KUKA KRL program: LOGO.src, LOGO.dat

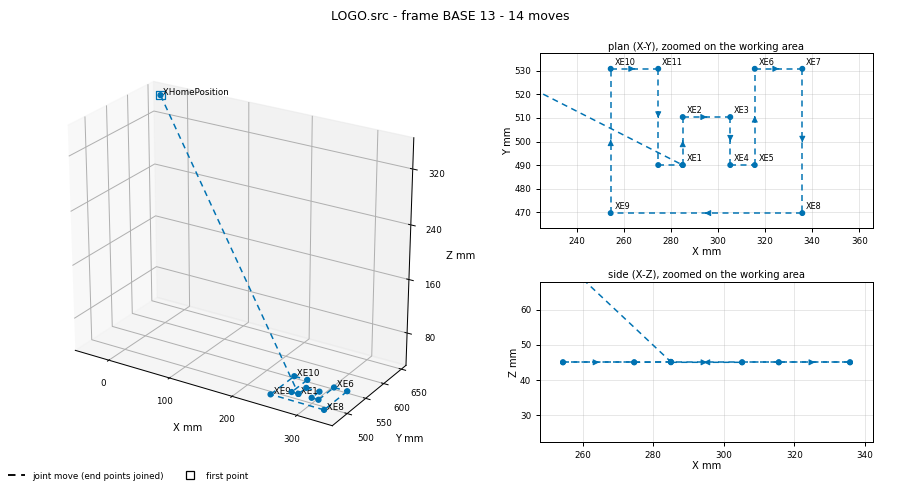
[picture p0: tool path of LOGO.src in frame BASE 13, 14 of 14 moves have a stored position in this frame; points joined in program order, loops and branches not executed]
--- LOGO.src ---
&ACCESS RVP
&REL 3
&PARAM EDITMASK = *
&PARAM TEMPLATE = C:\KRC\Roboter\Template\vorgabe

DEF LOGO( )
;FOLD INI;%{PE}
  ;FOLD BASISTECH INI
    GLOBAL INTERRUPT DECL 3 WHEN $STOPMESS==TRUE DO IR_STOPM ( )
    INTERRUPT ON 3
    BAS (#INITMOV,0 )
  ;ENDFOLD (BASISTECH INI)
  ;FOLD USER INI
    ;Make your modifications here

  ;ENDFOLD (USER INI)
;ENDFOLD (INI)


$BWDSTART=FALSE
PDAT_ACT=PPDAT1
FDAT_ACT=FHomePosition
BAS(#PTP_PARAMS,100)
PTP XHomePosition

$BWDSTART=FALSE
PDAT_ACT=PPDAT1
FDAT_ACT=FE1
BAS(#PTP_PARAMS,100)
PTP XE1
$BWDSTART=FALSE
PDAT_ACT=PPDAT1
FDAT_ACT=FE1
BAS(#PTP_PARAMS,100)
PTP XE2
$BWDSTART=FALSE
PDAT_ACT=PPDAT1
FDAT_ACT=FE1
BAS(#PTP_PARAMS,100)
PTP XE3
$BWDSTART=FALSE
PDAT_ACT=PPDAT1
FDAT_ACT=FE1
BAS(#PTP_PARAMS,100)
PTP XE4
$BWDSTART=FALSE
PDAT_ACT=PPDAT1
FDAT_ACT=FE1
BAS(#PTP_PARAMS,100)
PTP XE5
$BWDSTART=FALSE
PDAT_ACT=PPDAT1
FDAT_ACT=FE1
BAS(#PTP_PARAMS,100)
PTP XE6
$BWDSTART=FALSE
PDAT_ACT=PPDAT1
FDAT_ACT=FE1
BAS(#PTP_PARAMS,100)
PTP XE7
$BWDSTART=FALSE
PDAT_ACT=PPDAT1
FDAT_ACT=FE1
BAS(#PTP_PARAMS,100)
PTP XE8
$BWDSTART=FALSE
PDAT_ACT=PPDAT1
FDAT_ACT=FE1
BAS(#PTP_PARAMS,100)
PTP XE9
$BWDSTART=FALSE
PDAT_ACT=PPDAT1
FDAT_ACT=FE1
BAS(#PTP_PARAMS,100)
PTP XE10
$BWDSTART=FALSE
PDAT_ACT=PPDAT1
FDAT_ACT=FE1
BAS(#PTP_PARAMS,100)
PTP XE11
$BWDSTART=FALSE
PDAT_ACT=PPDAT1
FDAT_ACT=FE1
BAS(#PTP_PARAMS,100)
PTP XE12
$BWDSTART=FALSE
PDAT_ACT=PPDAT1
FDAT_ACT=FE1
BAS(#PTP_PARAMS,100)
PTP XE1
; Offset
;PTP {X 0,Y 0,Z 50,A 0,B 0,C 0} : XE1

END

--- LOGO.dat ---
&ACCESS RVP
&REL 3
&PARAM EDITMASK = *
&PARAM TEMPLATE = C:\KRC\Roboter\Template\vorgabe
DEFDAT  LOGO
;FOLD EXTERNAL DECLARATIONS;%{PE}%MKUKATPBASIS,%CEXT,%VCOMMON,%P
;FOLD BASISTECH EXT;%{PE}%MKUKATPBASIS,%CEXT,%VEXT,%P
EXT  BAS (BAS_COMMAND  :IN,REAL  :IN )
DECL INT SUCCESS
;ENDFOLD (BASISTECH EXT)
;FOLD USER EXT;%{E}%MKUKATPUSER,%CEXT,%VEXT,%P
;Make your modifications here

;ENDFOLD (USER EXT)
;ENDFOLD (EXTERNAL DECLARATIONS)
DECL BASIS_SUGG_T LAST_BASIS={POINT1[] "E12                      ",POINT2[] "E12                      ",CP_PARAMS[] "CPDAT0                  ",PTP_PARAMS[] "PDAT1                   ",CONT[] "                        ",CP_VEL[] "2.0                     ",PTP_VEL[] "100                     ",SYNC_PARAMS[] "SYNCDAT                 ",SPL_NAME[] "S0                      ",A_PARAMS[] "ADAT0                   "}
DECL E6POS XHOMEPOSITION={X -39.1373024,Y 654.730652,Z 349.722229,A 84.3230286,B -2.04451323,C 156.065094,S 6,T 26,E1 0.0,E2 0.0,E3 0.0,E4 0.0,E5 0.0,E6 0.0}

DECL FDAT FHomePosition={TOOL_NO 12,BASE_NO 13,IPO_FRAME #BASE,POINT2[] " ",TQ_STATE FALSE}
DECL PDAT PPDAT1={VEL 100.000,ACC 100.000,APO_DIST 100.000,APO_MODE #CDIS,GEAR_JERK 50.0000,EXAX_IGN 0}
DECL FDAT FE1={TOOL_NO 12,BASE_NO 13,IPO_FRAME #BASE,POINT2[] " ",TQ_STATE FALSE}

DECL E6POS XE1={X 285,Y 490,Z 45.187,A 75.7398453,B -0.472523630,C 166.038666,S 6,T 26,E1 0.0,E2 0.0,E3 0.0,E4 0.0,E5 0.0,E6 0.0}
DECL E6POS XE2={X 285,Y 510.4,Z 45.052,A 75.7398453,B -0.472523630,C 166.038666,S 6,T 26,E1 0.0,E2 0.0,E3 0.0,E4 0.0,E5 0.0,E6 0.0}
DECL E6POS XE3={X 305.2,Y 510.4,Z 45.0524,A 75.7398453,B -0.472523630,C 166.038666,S 6,T 26,E1 0.0,E2 0.0,E3 0.0,E4 0.0,E5 0.0,E6 0.0}
DECL E6POS XE4={X 305.2,Y 490,Z 45.0524,A 75.7398453,B -0.472523630,C 166.038666,S 6,T 26,E1 0.0,E2 0.0,E3 0.0,E4 0.0,E5 0.0,E6 0.0}
DECL E6POS XE5={X 315.6,Y 490,Z 45.0524,A 75.7398453,B -0.472523630,C 166.038666,S 6,T 26,E1 0.0,E2 0.0,E3 0.0,E4 0.0,E5 0.0,E6 0.0}
DECL E6POS XE6={X 315.6,Y 530.9,Z 45.0524,A 75.7398453,B -0.472523630,C 166.038666,S 6,T 26,E1 0.0,E2 0.0,E3 0.0,E4 0.0,E5 0.0,E6 0.0}
DECL E6POS XE7={X 335.8,Y 530.9,Z 45.0524,A 75.7398453,B -0.472523630,C 166.038666,S 6,T 26,E1 0.0,E2 0.0,E3 0.0,E4 0.0,E5 0.0,E6 0.0}
DECL E6POS XE8={X 335.8,Y 469.6,Z 45.0524,A 75.7398453,B -0.472523630,C 166.038666,S 6,T 26,E1 0.0,E2 0.0,E3 0.0,E4 0.0,E5 0.0,E6 0.0}
DECL E6POS XE9={X 254.4,Y 469.6,Z 45.0524,A 75.7398453,B -0.472523630,C 166.038666,S 6,T 26,E1 0.0,E2 0.0,E3 0.0,E4 0.0,E5 0.0,E6 0.0}
DECL E6POS XE10={X 254.4,Y 530.9,Z 45.0524,A 75.7398453,B -0.472523630,C 166.038666,S 6,T 26,E1 0.0,E2 0.0,E3 0.0,E4 0.0,E5 0.0,E6 0.0}
DECL E6POS XE11={X 274.6,Y 530.9,Z 45.0524,A 75.7398453,B -0.472523630,C 166.038666,S 6,T 26,E1 0.0,E2 0.0,E3 0.0,E4 0.0,E5 0.0,E6 0.0}
DECL E6POS XE12={X 274.6,Y 490,Z 45.0524,A 75.7398453,B -0.472523630,C 166.038666,S 6,T 26,E1 0.0,E2 0.0,E3 0.0,E4 0.0,E5 0.0,E6 0.0}

ENDDAT
